RoboDK station: simple_ur5e_station_cable_yanking.rdk

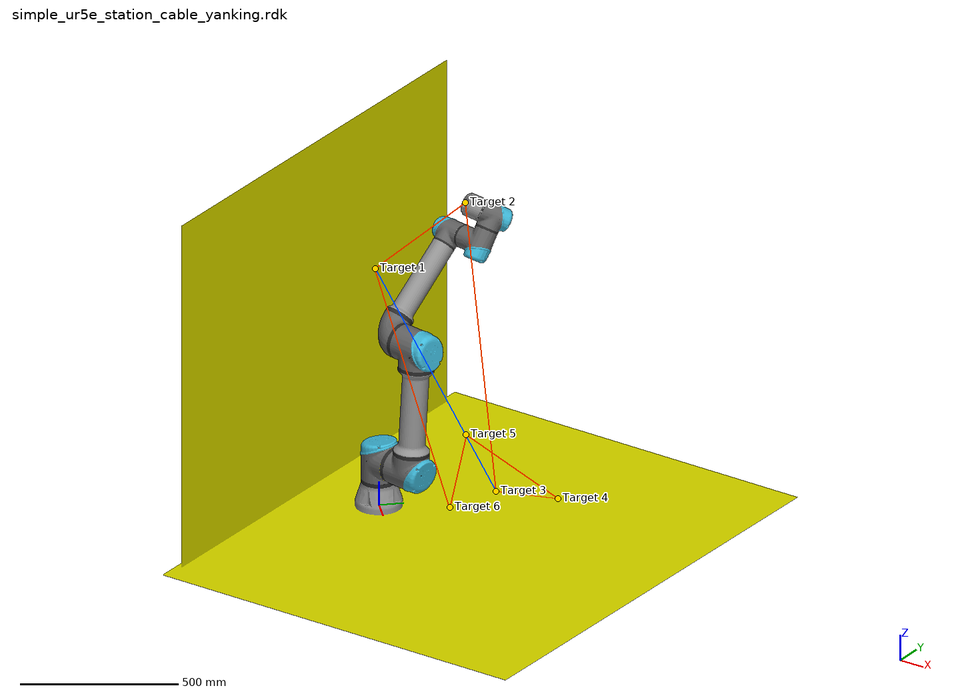
[picture v0: the station drawn from its stored meshes, robots at their saved joint values, targets as dots, program paths as lines]
Station simple_ur5e_station_cable_yanking_shorter. Poses are relative to the parent item; angles as X-Y-Z fixed-axis rotations.
Station parameters (name, value as stored): CollisionFreePlanner, UR5e, CollisionFreePlanner-Rob UR5e
  - frame UR5e Base at (0, 0, 0) mm, rotated rx 0 ry 0 rz -45 deg
    - robot UR5e: 6 axes, payload 5 kg, reach 850 mm, repeatability 0.03 mm, weight 18.4 kg
        modified DH rows (alpha deg, a mm, theta deg, d mm): 0, 0, 0, 162.5; 90, 0, 180, 0; 0, 425, 0, 0; 0, 392.25, 0, 133.3; -90, 0, 0, 99.7; 90, 0, 180, 99.6
        joint limits [-360, -360, -360, -360, -360, -360] to [360, 360, 360, 360, 360, 360]; home [0, -90, -90, 0, 90, 0]; saved at [125.728, -94.363, -43.442, -76.24, -122.946, 46.387]
    - target Target 1 (Cartesian target) at (270.26, -59.11, 963.67) mm, rotated rx -90 ry 54.09 rz -135 deg; joints [45, -90, -35.91, 0, 0, 0] of UR5e
    - target Target 2 (Cartesian target) at (-116.48, 297.46, 979.13) mm, rotated rx -36.77 ry 54.09 rz -135 deg; joints [125.728, -94.363, -43.442, -76.24, -122.946, 46.387] of UR5e
    - target Target 3 (Cartesian target) at (641.02, 261.87, 333.92) mm, rotated rx 160.83 ry 8.8 rz 64.71 deg; joints [36.34, -155.56, -10.93, 78.26, -69.05, 59.81] of UR5e
    - target Target 4 (Cartesian target) at (723.9, 446.23, 332.43) mm, rotated rx 138.75 ry 6.47 rz -120.79 deg; joints [36.34, -155.56, -10.93, -116.93, 129.82, 59.81] of UR5e
    - target Target 5 (Cartesian target) at (-270.8, 328.23, 88.26) mm, rotated rx 138.75 ry 6.47 rz -120.79 deg; joints [148.934, -129.854, -141.821, 43.121, 85.328, 175.515] of UR5e
    - target Target 6 (Cartesian target) at (613.58, 119.55, 274.82) mm, rotated rx -21.42 ry 4.17 rz 81.27 deg; joints [177.7, -28.54, 50.64, 46.96, -83.79, 175.51] of UR5e
    - target Target 7 (Cartesian target) at (270.26, -59.11, 963.67) mm, rotated rx -90 ry 54.09 rz -135 deg; joints [141.484, -105.404, 57.351, 228.053, -96.484, 54.09] of UR5e
  - object Floor at (0, 0, 0) mm, size 1320 x 1606 x 0.7 mm
  - object Back wall at (0, 0, 0) mm, rotated rx 0 ry -90 rz 0 deg, size 1200 x 1460 x 0.6 mm
  - object Front wall at (0, 0, 0) mm, rotated rx 0 ry -90 rz 0 deg, size 1200 x 1460 x 0.6 mm
  - object Right wall at (0, 0, 0) mm, size 1250 x 0.6 x 1200 mm
  - program Prog1 (9 instructions, listed below)
  - object Left wall at (0, 0, 0) mm, size 1250 x 0.6 x 1200 mm
  - program Cycle RDK (no cycle counting) (12 instructions, listed below)
  - Python program set_joint_speed (listed below)
  - program Target7ToTarget8 (2 instructions, listed below)
  - program Target8ToTarget1 (3 instructions, listed below)
  - program Target1ToTarget8 (3 instructions, listed below)
  - program Target8ToTarget9 (2 instructions, listed below)
  - Python program loopCycle (listed below)
  - program Cycle python (cycle counting) (1 instructions, listed below)
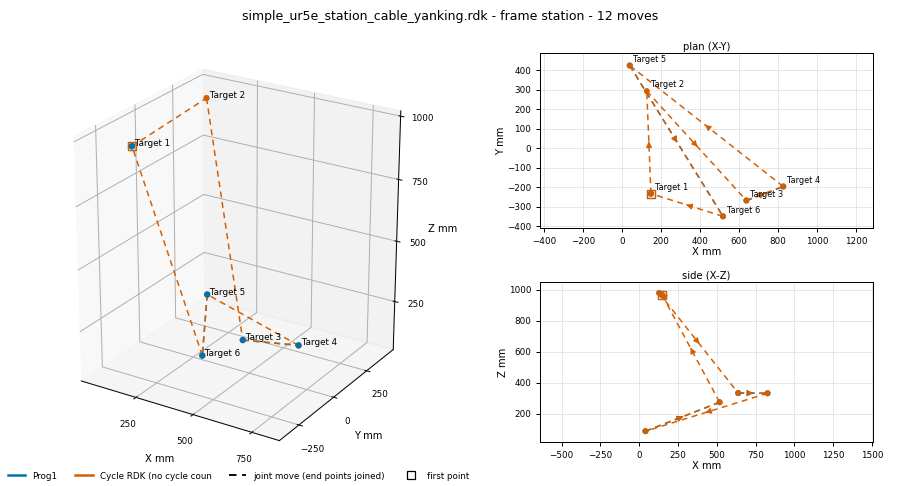
[picture p0: tool path of simple_ur5e_station_cable_yanking.rdk in frame station, 12 of 25 moves have a stored position in this frame; points joined in program order, loops and branches not executed]
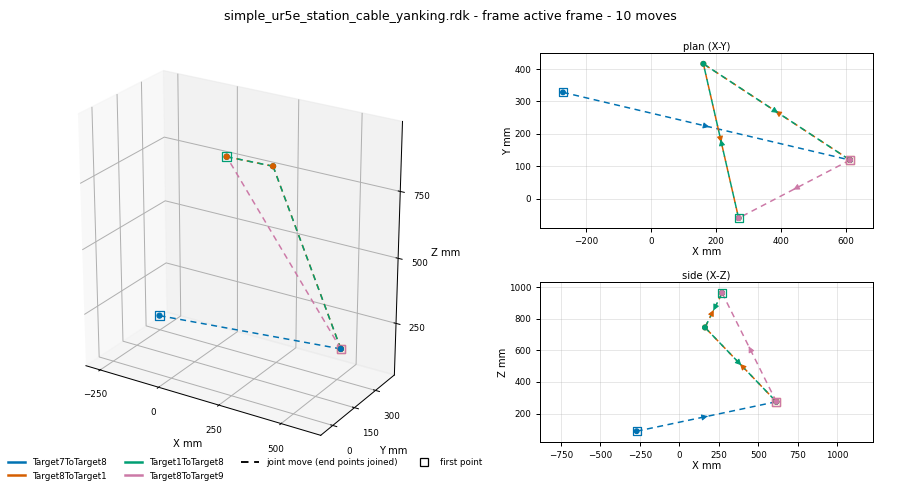
[picture p1: tool path of simple_ur5e_station_cable_yanking.rdk in frame active frame, 10 of 25 moves have a stored position in this frame; points joined in program order, loops and branches not executed]

--- program Prog1 (robot UR5e) ---
  Set Ref.: UR5e Base
  MoveJ (Target 1)
  MoveJ (Target 2) [its target is no longer in the station]
  MoveJ (Target 3) [its target is no longer in the station]
  MoveJ (Target 5) -> target Target 3
  MoveJ (Target 6) -> target Target 4
  MoveJ (Target 6) [its target is no longer in the station]
  MoveJ (Target 7) -> target Target 5
  MoveJ (Target 8) -> target Target 6

--- program Cycle RDK (no cycle counting) (robot UR5e) ---
  Set Ref.: UR5e Base
  Set speed (50.0 mm/s)
  MoveJ (Target 1)
  Smooth(50)
  MoveJ (Target 2)
  MoveJ (Target 3)
  Smooth(50)
  MoveJ (Target 4)
  MoveJ (Target 5)
  MoveJ (Target 6)
  MoveJ (Target 7)
  Smooth(30)

--- Python program set_joint_speed ---
from robolink import *
from robodk import *

RDK = Robolink()
robot = RDK.Item('UR5e', ITEM_TYPE_ROBOT)
robot.setSpeedJoints(45)

--- program Target7ToTarget8 (robot UR5e) ---
  MoveJ (Pt 1 (S101)) to (-270.8, 328.23, 88.26) mm, rotated rx 138.75 ry 6.47 rz -120.79 deg; joints [148.934, -129.854, -141.821, 43.121, 85.328, 175.515]
  MoveJ (Pt 2 (S102)) to (613.58, 119.55, 274.82) mm, rotated rx -21.42 ry 4.17 rz 81.27 deg; joints [177.7, -28.54, 50.64, 46.96, -83.79, 175.51]

--- program Target8ToTarget1 (robot UR5e) ---
  MoveJ (Pt 1 (S102)) to (613.58, 119.55, 274.82) mm, rotated rx -21.42 ry 4.17 rz 81.27 deg; joints [177.7, -28.54, 50.64, 46.96, -83.79, 175.51]
  MoveJ (Pt 2 (S95)) to (161.76, 416.07, 745.11) mm, rotated rx -96.43 ry 24.01 rz -131.02 deg; joints [244.058, -48.052, -21.15, 43.714, -166.254, 179.293]
  MoveJ (Pt 3 (S103)) to (270.26, -59.11, 963.67) mm, rotated rx -90 ry 54.09 rz -135 deg; joints [45, -90, -35.91, 0, 0, 0]

--- program Target1ToTarget8 (robot UR5e) ---
  MoveJ (Pt 1 (S103)) to (270.26, -59.11, 963.67) mm, rotated rx -90 ry 54.09 rz -135 deg; joints [45, -90, -35.91, 0, 0, 0]
  MoveJ (Pt 2 (S95)) to (161.76, 416.07, 745.11) mm, rotated rx -96.43 ry 24.01 rz -131.02 deg; joints [244.058, -48.052, -21.15, 43.714, -166.254, 179.293]
  MoveJ (Pt 3 (S102)) to (613.58, 119.55, 274.82) mm, rotated rx -21.42 ry 4.17 rz 81.27 deg; joints [177.7, -28.54, 50.64, 46.96, -83.79, 175.51]

--- program Target8ToTarget9 (robot UR5e) ---
  MoveJ (Pt 1 (S102)) to (613.58, 119.55, 274.82) mm, rotated rx -21.42 ry 4.17 rz 81.27 deg; joints [177.7, -28.54, 50.64, 46.96, -83.79, 175.51]
  MoveJ (Pt 2 (S104)) to (270.26, -59.11, 963.67) mm, rotated rx -90 ry 54.09 rz -135 deg; joints [141.484, -105.404, 57.351, 228.053, -96.484, 54.09]

--- Python program loopCycle ---
from robolink import *
from robodk import *
from datetime import datetime

timestamp = datetime.now()
filename = "cycle_count_" + timestamp.strftime("%d_%m_%Y_%H_%M_%S")+".txt"
path = "/home/melyso/Documents/python_scripts/cycle_counts/" + filename
fo = open(path, "w")
fo.write("0")
fo.close()

joint_speed = 45 #in deg/s
target_count = 7

RDK = Robolink()
robot = RDK.Item('UR5e', ITEM_TYPE_ROBOT)

#Acquire targets in list
targets = []
for i in range(0,target_count):
        targets.append(RDK.Item('Target ' + str(i+1)))

robot.setSpeedJoints(joint_speed)

while True:
        for t in targets:
                robot.MoveJ(t)

        fo = open(path, "r")
        cycle_count = int(fo.read())
        fo.close()
        cycle_count += 1
        fo = open(path, "w")
        fo.write(str(cycle_count))
        fo.close()

--- program Cycle python (cycle counting) (robot UR5e) ---
  Call loopCycle
